// TIA Portal project "iodevice" (V15)

(* hardware
DEVICE "S71500/ET200MP station_1"  S7-1500 station
   slot 0: "Rail_0"  Rack  6ES7 590-1***0-0AA0
   slot 1: "PLC_1"  CPU 1511-1 PN  6ES7 511-1AK00-0AB0  V1.8
      slot 3: "CPU display_1"  6ES7591-1AA00-0AA0
   slot 2: "AI/AQ 4xU/I/RTD/TC / 2xU/I ST_1"  AI/AQ 4xU/I/RTD/TC / 2xU/I ST  6ES7 534-7QE00-0AB0  V1.0
*)

// ===== PLC "PLC_1"  CPU 1511-1 PN =====

VAR_GLOBAL   // PLC tag table "Default tag table"
   "trigger" AT %Q0.0 : Bool;
   "output" AT %Q0.1 : Bool;
   "inturpt" AT %Q0.2 : Bool;
   "genIN" AT %Q0.3 : Bool;
   "genOUT" AT %Q0.4 : Bool;
   "in1" AT %M0.0 : Bool;
   "out1" AT %M0.1 : Bool;
   "out2" AT %M0.2 : Bool;
   "out3" AT %M0.3 : Bool;
   "out3count" AT %MW2 : Int;
   "out1count" AT %MW4 : Int;
   "t1out" AT %M0.4 : Bool;
   "t2out" AT %M0.5 : Bool;
   "t3out" AT %M0.6 : Bool;
   "t4out" AT %M0.7 : Bool;
   "et4" AT %MD6 : Time;
   "et3" AT %MD10 : DWord;
   "et2" AT %MD14 : DWord;
   "et1" AT %MD18 : DInt;
   "timerswitch" AT %M1.0 : Bool;
   "timerswitch(1)" AT %M1.1 : Bool;
   "timerswitch(2)" AT %M1.2 : Bool;
   "timereset" AT %M1.3 : Bool;
END_VAR

// folder: System blocks/Program resources

DATA_BLOCK "pulse"   // DB1
{ S7_Optimized_Access := 'TRUE' }
AUTHOR : Simatic
FAMILY : IEC
NAME : IEC_TMR
VERSION : 1.0
// stored: InstanceOfName IEC_TIMER
"IEC_TIMER"
BEGIN
END_DATA_BLOCK

DATA_BLOCK "ton"   // DB2
{ S7_Optimized_Access := 'TRUE' }
AUTHOR : Simatic
FAMILY : IEC
NAME : IEC_TMR
VERSION : 1.0
// stored: InstanceOfName IEC_TIMER
"IEC_TIMER"
BEGIN
END_DATA_BLOCK

DATA_BLOCK "tof"   // DB3
{ S7_Optimized_Access := 'TRUE' }
AUTHOR : Simatic
FAMILY : IEC
NAME : IEC_TMR
VERSION : 1.0
// stored: InstanceOfName IEC_TIMER
"IEC_TIMER"
BEGIN
END_DATA_BLOCK

DATA_BLOCK "tonr"   // DB4
{ S7_Optimized_Access := 'TRUE' }
AUTHOR : Simatic
FAMILY : IEC
NAME : IEC_TMR
VERSION : 1.0
// stored: InstanceOfName IEC_TIMER
"IEC_TIMER"
BEGIN
END_DATA_BLOCK

// folder: (top level)

ORGANIZATION_BLOCK "Main"   // OB1, LAD, ProgramCycle
TITLE = "Main Program Sweep (Cycle)"
{ S7_Optimized_Access := 'TRUE' }
VERSION : 0.1
   VAR_INPUT
      Initial_Call : Bool;   // Initial call of this OB
      Remanence : Bool;   // =True, if remanent data are available
   END_VAR
BEGIN

REGION Network 1
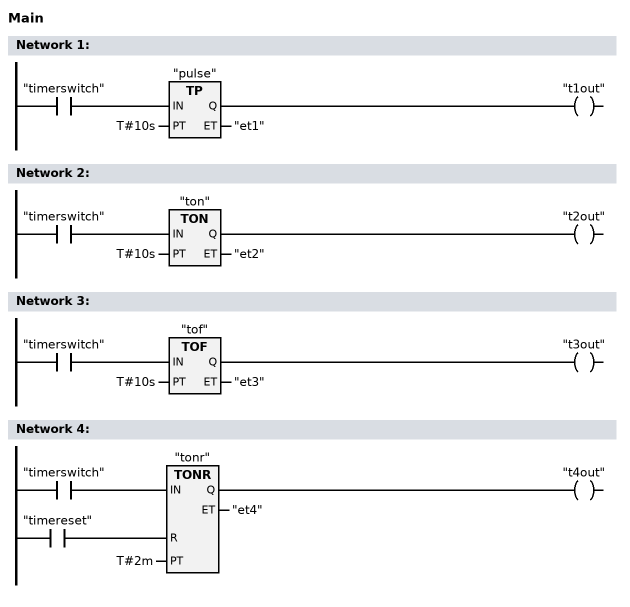
   "pulse".TP(IN := "timerswitch", PT := T#10s, ET => "et1");
   "t1out" := "pulse".Q;
END_REGION

REGION Network 2
   "ton".TON(IN := "timerswitch", PT := T#10s, ET => "et2");
   "t2out" := "ton".Q;
END_REGION

REGION Network 3
   "tof".TOF(IN := "timerswitch", PT := T#10s, ET => "et3");
   "t3out" := "tof".Q;
END_REGION

REGION Network 4
   "tonr".TONR(IN := "timerswitch", R := "timereset", PT := T#2m, ET => "et4");
   "t4out" := "tonr".Q;
END_REGION
END_ORGANIZATION_BLOCK